// Interface to implement when requiring AMS address
INTERFACE I_RequiresAmsAddress

// Gets or sets the Ams address structure
PROPERTY AmsAddress : REFERENCE TO Tc2_System.ST_AmsAddr
GET
END_GET
SET
END_SET
END_PROPERTY

END_INTERFACE

(* stored: Version 1.1.0.1, ProductVersion 3.1.4024.13
   Itf I_RequiresAmsAddress: Id {15ae4c03-32d8-07b8-0d05-f15d9cda81b9}
   Property AmsAddress: Id {66a0c4a6-c5be-0e29-1c2e-325d469fedba}
   Get Get: Id {8585a222-f138-096f-3db9-1290193c7115}
   Set Set: Id {636597e4-a45e-0f16-1b2e-b0c9337969de} *)
